// TIA Portal project "Palletizer_TIA_Portal" (V16)

(* hardware
DEVICE "S7-1200 station_1"  S7-1200 Station
   slot 0: "Rack_0"  S7-1200 Rack  Rack  V1.0
   slot 1: "PLC_1"  CPU 1215C DC/DC/DC  6ES7 215-1AG40-0XB0  V4.4
   slot 2: "DI 8x24VDC_1"  6ES7 221-1BF32-0XB0  V2.0
*)

// ===== PLC "PLC_1"  CPU 1215C DC/DC/DC =====

VAR_GLOBAL   // PLC tag table "Tabla de variables estándar"
   "Tag_9" AT %M10.6 : Bool;
   "flanco_p_sensor_entrada_cajas" AT %M10.7 : Bool;
   "Reset_contador_1" AT %M11.0 : Bool;
   "Tag_11" AT %M500.0 : Bool;
   "flanco_p_sensor_ascensor_pales" AT %M11.5 : Bool;
END_VAR

VAR_GLOBAL   // PLC tag table "Entradas"
   "Pallet_at_entry" AT %I0.0 : Bool;   // Sensor al final del transportador de rodillos alimentador, justo antes de la paletizadora
   "Pallet_at_exit" AT %I0.1 : Bool;   // Sensor a la entrada del transportador de rodillos de salida, justo despues de la paletizadora
   "Pallet_loaded" AT %I0.2 : Bool;   // Sensor dentro de la paletizadora, indica que el pale esta dentro
   "Box_at_entry" AT %I0.3 : Bool;   // Sensor al final de la cinta alimentadora de cajas
   "Pusher_limit" AT %I0.4 : Bool;   // Sensor que indica que el empujador esta en alguna de sus posiciones limite
   "Plate_limit" AT %I0.5 : Bool;   // Sensor que indica que la ventana esta en alguna de sus posiciones limite, completamente abierta o completamente cerrada
   "Clamped" AT %I0.6 : Bool;   // Sensor que indica que la mordaza está cerrada
   "Elevator_moving" AT %I0.7 : Bool;   // Sensor que indica que el ascensor está en movimiento
   "Start" AT %I1.0 : Bool;   // Pulsador de start
   "Reset" AT %I1.1 : Bool;   // Pulsador de reset
   "Stop" AT %I1.2 : Bool;   // Pulsador de stop
   "Emergency_stop" AT %I1.3 : Bool;   // Seta de emergencia
   "Auto" AT %I1.4 : Bool;   // Conmutador en modo automatico
   "Manual" AT %I1.5 : Bool;   // Conmutador en modo manual
END_VAR

VAR_GLOBAL   // PLC tag table "Salidas"
   "Pallet_feeder" AT %Q0.0 : Bool;   // Transportador de rodillos alimentador de pales
   "Load_pallet" AT %Q0.1 : Bool;   // Transportador dentro del paletizador
   "Exit_conveyor" AT %Q0.2 : Bool;   // Transportador de rodillos de salida
   "Move_to_limit" AT %Q0.3 : Bool;   // Salida booleana para hacer que la subida o bajada del ascensor sea entre el limite inferior y superior en un solo movimiento
   "Elevator_up" AT %Q0.4 : Bool;   // Ascensor arriba
   "Elevator_down" AT %Q0.5 : Bool;   // Ascensor abajo
   "Box_feeder" AT %Q0.6 : Bool;   // Cinta alimentadora de cajas
   "Turn" AT %Q0.7 : Bool;   // Empujador para girar la caja
   "Push" AT %Q1.0 : Bool;   // Empujador de la caja de la cinta hacia la ventana
   "Load_belt" AT %Q1.1 : Bool;   // Cinta de carga delas cajas dentro del paletizador
   "Clamp" AT %Q1.2 : Bool;   // Mordaza para compactar las cajas
   "Open_plate" AT %Q1.3 : Bool;   // Abrir/cerrar ventana
   "Warning_light" AT %Q1.4 : Bool;   // Luz de peligro
   "Start_light" AT %Q1.5 : Bool;   // Luz de boton de start
   "Reset_light" AT %Q1.6 : Bool;   // Luz de boton de reset
   "Stop_light" AT %Q1.7 : Bool;   // Luz de boton de stop
END_VAR

VAR_GLOBAL   // PLC tag table "variables_en_memoria"
   "Pallet_feeder_manual" AT %M100.0 : Bool;   // Transportador de rodillos alimentador de pales
   "Load_pallet_manual" AT %M100.1 : Bool;   // Transportador dentro del paletizador
   "Exit_conveyor_manual" AT %M100.2 : Bool;   // Transportador de rodillos de salida
   "Move_to_limit_manual" AT %M100.3 : Bool;   // Salida booleana para hacer que la subida o bajada del ascensor sea entre el limite inferior y superior en un solo movimiento
   "Elevator_up_manual" AT %M100.4 : Bool;   // Ascensor arriba
   "Elevator_down_manual" AT %M100.5 : Bool;   // Ascensor abajo
   "Box_feeder_manual" AT %M100.6 : Bool;   // Cinta alimentadora de cajas
   "Turn_manual" AT %M100.7 : Bool;   // Empujador para girar la caja
   "Push_manual" AT %M101.0 : Bool;   // Empujador de la caja de la cinta hacia la ventana
   "Load_belt_manual" AT %M101.1 : Bool;   // Cinta de carga delas cajas dentro del paletizador
   "Clamp_manual" AT %M101.2 : Bool;   // Mordaza para compactar las cajas
   "Open_plate_manual" AT %M101.3 : Bool;   // Abrir/cerrar ventana
   "marcha" AT %M0.0 : Bool;
   "modo_cambiado" AT %M0.1 : Bool;
   "Pallet_terminado" AT %M0.2 : Bool;
   "aux1" AT %M0.3 : Bool;
   "paletizadora_libre" AT %M0.4 : Bool;
   "pale_terminado" AT %M0.5 : Bool;
   "primer_nivel_OK" AT %M0.6 : Bool;
   "segundo_nivel_OK" AT %M0.7 : Bool;
   "flanco_n_sensor_entrada_pales" AT %M10.0 : Bool;
   "flanco_p_sensor_entrada_pales" AT %M10.1 : Bool;
   "flanco_n_sensor_ascensor_pales" AT %M10.3 : Bool;
   "flanco_n_sensor_salida_pales" AT %M10.4 : Bool;
   "flanco_p_sensor_ascensor_pales(1)" AT %M10.5 : Bool;
   "flanco_selector_modo_manual" AT %M200.0 : Bool;
   "flanco_selector_modo_auto" AT %M200.1 : Bool;
   "numero_cajas_1" AT %MW2 : Int;
   "numero_cajas_2" AT %MW4 : Int;
   "numero_columnas-1" AT %MW6 : Int;
   "numero_filas" AT %MW8 : Int;
END_VAR

DATA_BLOCK "control_ascensor_DB"   // DB2
{ S7_Optimized_Access := 'TRUE' }
VERSION : 0.1
// stored: InstanceOfName control_ascensor
"control_ascensor"
BEGIN
END_DATA_BLOCK

DATA_BLOCK "modo_automatico_DB"   // DB3
{ S7_Optimized_Access := 'TRUE' }
VERSION : 0.1
// stored: InstanceOfName modo_automatico
"modo_automatico"
BEGIN
END_DATA_BLOCK

FUNCTION_BLOCK "modo_automatico"   // FB2, LAD
{ S7_Optimized_Access := 'TRUE' }
VERSION : 0.1
   VAR
      E0 : Bool;
      E1 : Bool;
      E2 : Bool;
      E3 : Bool;
      E4 : Bool;
      E5 : Bool;
      "control_roller_1.1" : "control_roller_1";
      "control_roller_2.1" : "control_roller_2";
      control_ascensor_Instance : "control_ascensor";
      control_apilamiento_Instance : "control_apilamiento";
   END_VAR
   VAR_TEMP   // added for the SCL form of the ladder/FBD networks
      _w1 : Bool;
   END_VAR
BEGIN

REGION Network 1
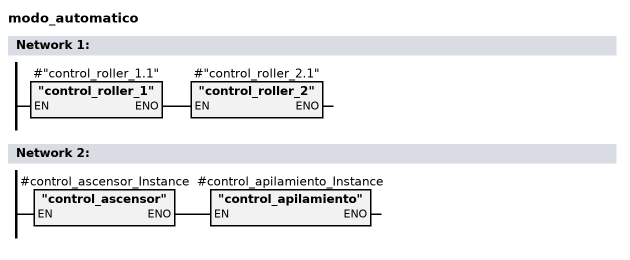
   RUNG wire#powerrail
      #"control_roller_1.1"()
      #"control_roller_2.1"()
   END_RUNG
   // the same network as SCL:
   #"control_roller_1.1"(ENO => #_w1);   // "control_roller_1"
   IF #_w1 THEN
       #"control_roller_2.1"();   // "control_roller_2"
   END_IF;
END_REGION

REGION Network 2
   RUNG wire#powerrail
      #control_ascensor_Instance()
      #control_apilamiento_Instance()
   END_RUNG
   // the same network as SCL:
   #control_ascensor_Instance(ENO => #_w1);   // "control_ascensor"
   IF #_w1 THEN
       #control_apilamiento_Instance();   // "control_apilamiento"
   END_IF;
END_REGION
END_FUNCTION_BLOCK

FUNCTION_BLOCK "control_roller_1"   // FB3, LAD
{ S7_Optimized_Access := 'TRUE' }
VERSION : 0.1
   VAR
      E1 : Bool;
      E2 : Bool;
      E3 : Bool;
      E4 : Bool;
      E5 : Bool;
      E0 : Bool;
   END_VAR
   VAR_TEMP   // added for the SCL form of the ladder/FBD networks
      _w1 : Bool;
      _w2 : Bool;
      _w3 : Bool;
      _w4 : Bool;
   END_VAR
BEGIN

REGION Network 1
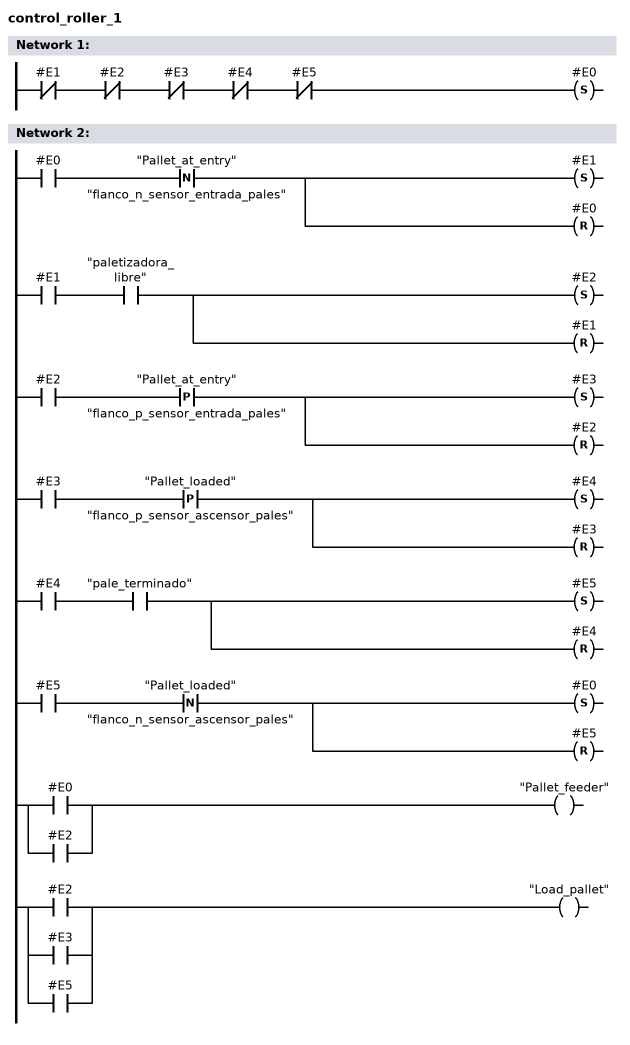
   RUNG wire#powerrail
      I_Contact( #E1 )
      I_Contact( #E2 )
      I_Contact( #E3 )
      I_Contact( #E4 )
      I_Contact( #E5 )
      S_Coil( #E0 )
   END_RUNG
   // the same network as SCL:
   IF NOT #E1 AND NOT #E2 AND NOT #E3 AND NOT #E4 AND NOT #E5 THEN #E0 := TRUE; END_IF;
END_REGION

REGION Network 2
   RUNG wire#powerrail
      Contact( #E0 )
      N_Contact(operand := "Pallet_at_entry", bit := "flanco_n_sensor_entrada_pales")
      wire#w1
      S_Coil( #E1 )
   END_RUNG
   RUNG wire#w1
      R_Coil( #E0 )
   END_RUNG
   RUNG wire#powerrail
      Contact( #E1 )
      Contact( "paletizadora_libre" )
      wire#w2
      S_Coil( #E2 )
   END_RUNG
   RUNG wire#w2
      R_Coil( #E1 )
   END_RUNG
   RUNG wire#powerrail
      Contact( #E2 )
      P_Contact(operand := "Pallet_at_entry", bit := "flanco_p_sensor_entrada_pales")
      wire#w3
      S_Coil( #E3 )
   END_RUNG
   RUNG wire#w3
      R_Coil( #E2 )
   END_RUNG
   RUNG wire#powerrail
      Contact( #E3 )
      P_Contact(operand := "Pallet_loaded", bit := "flanco_p_sensor_ascensor_pales")
      wire#w4
      S_Coil( #E4 )
   END_RUNG
   RUNG wire#w4
      R_Coil( #E3 )
   END_RUNG
   RUNG wire#powerrail
      Contact( #E4 )
      Contact( "pale_terminado" )
      wire#w5
      S_Coil( #E5 )
   END_RUNG
   RUNG wire#w5
      R_Coil( #E4 )
   END_RUNG
   RUNG wire#powerrail
      Contact( #E5 )
      N_Contact(operand := "Pallet_loaded", bit := "flanco_n_sensor_ascensor_pales")
      wire#w6
      S_Coil( #E0 )
   END_RUNG
   RUNG wire#w6
      R_Coil( #E5 )
   END_RUNG
   RUNG wire#powerrail
      Contact( #E0 )
      wire#w7
      Coil( "Pallet_feeder" )
   END_RUNG
   RUNG wire#powerrail
      Contact( #E2 )
   END_RUNG wire#w7
   RUNG wire#powerrail
      Contact( #E2 )
      wire#w8
      Coil( "Load_pallet" )
   END_RUNG
   RUNG wire#powerrail
      Contact( #E3 )
   END_RUNG wire#w8
   RUNG wire#powerrail
      Contact( #E5 )
   END_RUNG wire#w8
   // the same network as SCL:
   #_w1 := #E0 AND NOT "Pallet_at_entry" AND "flanco_n_sensor_entrada_pales";   // falling edge of "Pallet_at_entry"
   "flanco_n_sensor_entrada_pales" := "Pallet_at_entry";
   IF #_w1 THEN
       #E1 := TRUE;
       #E0 := FALSE;
   END_IF;
   IF #E1 AND "paletizadora_libre" THEN
       #E2 := TRUE;
       #E1 := FALSE;
   END_IF;
   #_w2 := #E2 AND "Pallet_at_entry" AND NOT "flanco_p_sensor_entrada_pales";   // rising edge of "Pallet_at_entry"
   "flanco_p_sensor_entrada_pales" := "Pallet_at_entry";
   IF #_w2 THEN
       #E3 := TRUE;
       #E2 := FALSE;
   END_IF;
   #_w3 := #E3 AND "Pallet_loaded" AND NOT "flanco_p_sensor_ascensor_pales";   // rising edge of "Pallet_loaded"
   "flanco_p_sensor_ascensor_pales" := "Pallet_loaded";
   IF #_w3 THEN
       #E4 := TRUE;
       #E3 := FALSE;
   END_IF;
   IF #E4 AND "pale_terminado" THEN
       #E5 := TRUE;
       #E4 := FALSE;
   END_IF;
   #_w4 := #E5 AND NOT "Pallet_loaded" AND "flanco_n_sensor_ascensor_pales";   // falling edge of "Pallet_loaded"
   "flanco_n_sensor_ascensor_pales" := "Pallet_loaded";
   IF #_w4 THEN
       #E0 := TRUE;
       #E5 := FALSE;
   END_IF;
   "Pallet_feeder" := #E0 OR #E2;
   "Load_pallet" := #E2 OR #E3 OR #E5;
END_REGION
END_FUNCTION_BLOCK

FUNCTION_BLOCK "control_roller_2"   // FB4, LAD
{ S7_Optimized_Access := 'TRUE' }
VERSION : 0.1
   VAR
      Timer_TP_1 : TP_TIME;
   END_VAR
   VAR_TEMP   // added for the SCL form of the ladder/FBD networks
      _w1 : Bool;
   END_VAR
BEGIN

REGION Network 1: Transportador de rodillos de salida
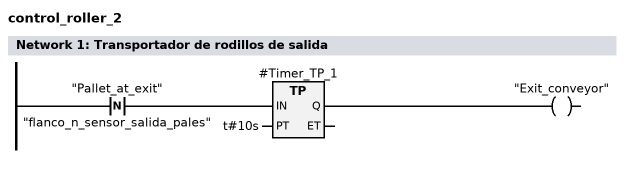
   #_w1 := NOT "Pallet_at_exit" AND "flanco_n_sensor_salida_pales";   // falling edge of "Pallet_at_exit"
   "flanco_n_sensor_salida_pales" := "Pallet_at_exit";
   #Timer_TP_1(IN := #_w1, PT := t#10s);   // TP
   "Exit_conveyor" := #Timer_TP_1.Q;
END_REGION
END_FUNCTION_BLOCK

FUNCTION_BLOCK "control_ascensor"   // FB5, LAD
{ S7_Optimized_Access := 'TRUE' }
VERSION : 0.1
   VAR
      E0 : Bool;
      E1 : Bool;
      E2 : Bool;
      E3 : Bool;
      E4 : Bool;
      E5 : Bool;
      E6 : Bool;
      TON_instancia_1 : TON_TIME;
      TON_instancia_2 : TON_TIME;
      TON_instancia_3 : TON_TIME;
   END_VAR
   VAR_TEMP   // added for the SCL form of the ladder/FBD networks
      _w1 : Bool;
      _w2 : Bool;
      _w3 : Bool;
      _w4 : Bool;
   END_VAR
BEGIN

REGION Network 1
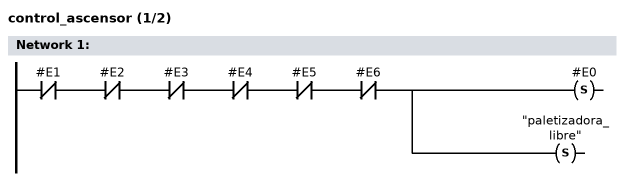
   RUNG wire#powerrail
      I_Contact( #E1 )
      I_Contact( #E2 )
      I_Contact( #E3 )
      I_Contact( #E4 )
      I_Contact( #E5 )
      I_Contact( #E6 )
      wire#w1
      S_Coil( #E0 )
   END_RUNG
   RUNG wire#w1
      S_Coil( "paletizadora_libre" )
   END_RUNG
   // the same network as SCL:
   IF NOT #E1 AND NOT #E2 AND NOT #E3 AND NOT #E4 AND NOT #E5 AND NOT #E6 THEN
       #E0 := TRUE;
       "paletizadora_libre" := TRUE;
   END_IF;
END_REGION

REGION Network 2: Salida booleana para hacer que la subida o bajada del ascensor sea entre el limite inferior y superior en un solo movimiento
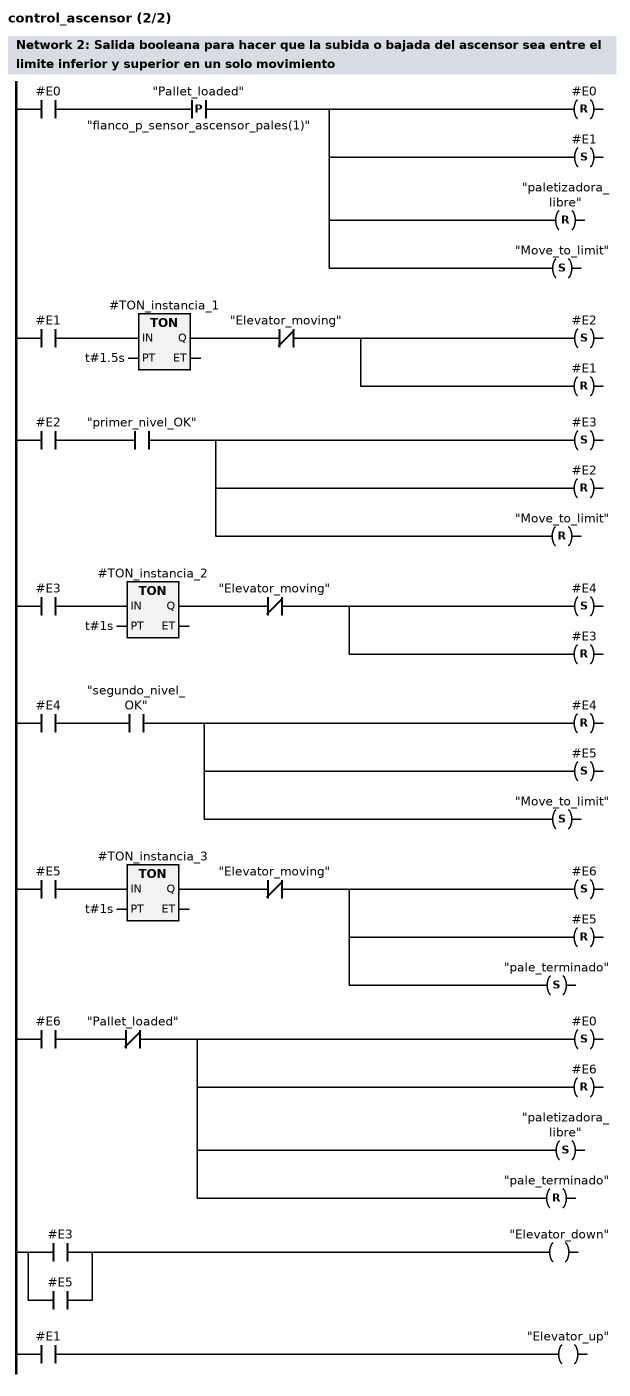
   #_w1 := #E0 AND "Pallet_loaded" AND NOT "flanco_p_sensor_ascensor_pales(1)";   // rising edge of "Pallet_loaded"
   "flanco_p_sensor_ascensor_pales(1)" := "Pallet_loaded";
   IF #_w1 THEN
       #E0 := FALSE;
       #E1 := TRUE;
       "paletizadora_libre" := FALSE;
       "Move_to_limit" := TRUE;
   END_IF;
   #TON_instancia_1(IN := #E1, PT := t#1.5s);   // TON
   IF #TON_instancia_1.Q AND NOT "Elevator_moving" THEN
       #E2 := TRUE;
       #E1 := FALSE;
   END_IF;
   IF #E2 AND "primer_nivel_OK" THEN #E3 := TRUE; END_IF;
   #_w2 := #E2 AND "primer_nivel_OK";
   IF #_w2 THEN
       #E2 := FALSE;
       "Move_to_limit" := FALSE;
   END_IF;
   #TON_instancia_2(IN := #E3, PT := t#1s);   // TON
   IF #TON_instancia_2.Q AND NOT "Elevator_moving" THEN
       #E4 := TRUE;
       #E3 := FALSE;
   END_IF;
   #_w3 := #E4 AND "segundo_nivel_OK";
   IF #_w3 THEN
       #E4 := FALSE;
       #E5 := TRUE;
       "Move_to_limit" := TRUE;
   END_IF;
   #TON_instancia_3(IN := #E5, PT := t#1s);   // TON
   IF #TON_instancia_3.Q AND NOT "Elevator_moving" THEN
       #E6 := TRUE;
       #E5 := FALSE;
       "pale_terminado" := TRUE;
   END_IF;
   IF #E6 AND NOT "Pallet_loaded" THEN #E0 := TRUE; END_IF;
   #_w4 := #E6 AND NOT "Pallet_loaded";
   IF #_w4 THEN
       #E6 := FALSE;
       "paletizadora_libre" := TRUE;
       "pale_terminado" := FALSE;
   END_IF;
   "Elevator_down" := #E3 OR #E5;
   "Elevator_up" := #E1;
END_REGION
END_FUNCTION_BLOCK

FUNCTION_BLOCK "control_apilamiento"   // FB6, LAD
{ S7_Optimized_Access := 'TRUE' }
VERSION : 0.1
   VAR
      E0 : Bool;
      E1 : Bool;
      E2 : Bool;
      E3 : Bool;
      E4 : Bool;
      E5 : Bool;
      E6 : Bool;
      E7 : Bool;
      E8 : Bool;
      E9 : Bool;
   END_VAR
   VAR RETAIN
      CTU_1 : CTD_INT;
   END_VAR
   VAR
      TON_1 : TON_TIME;
      TON_2 : TON_TIME;
      TON_3 : TON_TIME;
   END_VAR
   VAR RETAIN
      CTU_2 : CTU_INT;
   END_VAR
   VAR
      TON_4 : TON_TIME;
      TON_5 : TON_TIME;
      TON_6 : TON_TIME;
      TON_7 : TON_TIME;
      TON_8 : TON_TIME;
   END_VAR
   VAR_TEMP   // added for the SCL form of the ladder/FBD networks
      _w1 : Bool;
      _w2 : Bool;
      _w3 : Bool;
      _w4 : Bool;
   END_VAR
BEGIN

REGION Network 1
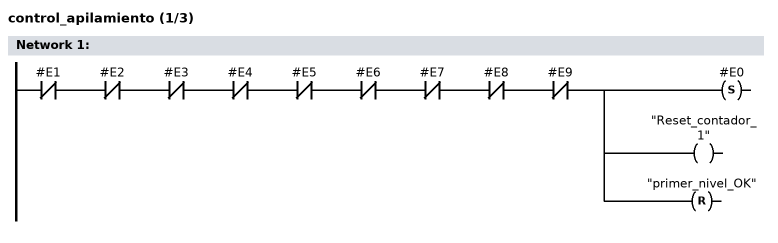
   RUNG wire#powerrail
      I_Contact( #E1 )
      I_Contact( #E2 )
      I_Contact( #E3 )
      I_Contact( #E4 )
      I_Contact( #E5 )
      I_Contact( #E6 )
      I_Contact( #E7 )
      I_Contact( #E8 )
      I_Contact( #E9 )
      wire#w1
      S_Coil( #E0 )
   END_RUNG
   RUNG wire#w1
      Coil( "Reset_contador_1" )
   END_RUNG
   RUNG wire#w1
      R_Coil( "primer_nivel_OK" )
   END_RUNG
   // the same network as SCL:
   #_w1 := NOT #E1 AND NOT #E2 AND NOT #E3 AND NOT #E4 AND NOT #E5 AND NOT #E6 AND NOT #E7 AND NOT #E8 AND NOT #E9;
   IF #_w1 THEN #E0 := TRUE; END_IF;
   "Reset_contador_1" := #_w1;
   IF #_w1 THEN "primer_nivel_OK" := FALSE; END_IF;
END_REGION

REGION Network 2
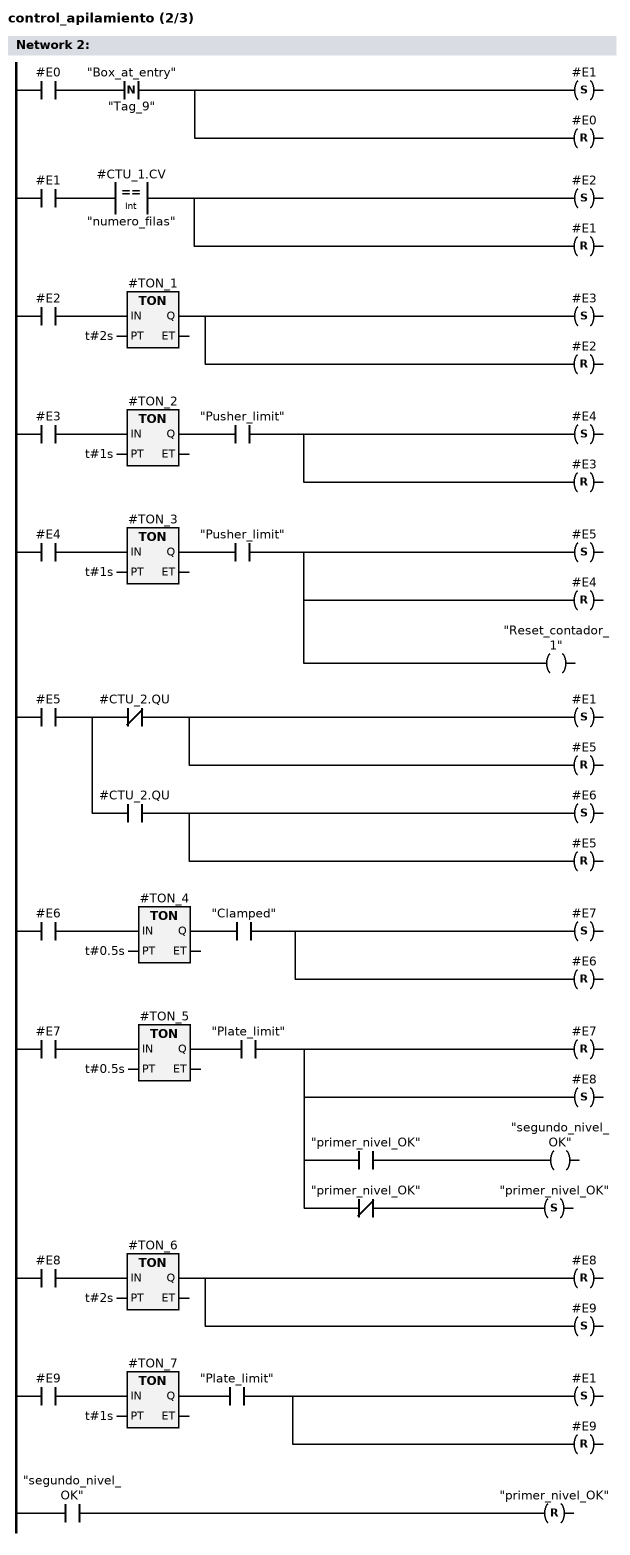
   #_w1 := #E0 AND NOT "Box_at_entry" AND "Tag_9";   // falling edge of "Box_at_entry"
   "Tag_9" := "Box_at_entry";
   IF #_w1 THEN
       #E1 := TRUE;
       #E0 := FALSE;
   END_IF;
   IF #E1 AND (#CTU_1.CV = "numero_filas") THEN
       #E2 := TRUE;
       #E1 := FALSE;
   END_IF;
   #TON_1(IN := #E2, PT := t#2s);   // TON
   IF #TON_1.Q THEN
       #E3 := TRUE;
       #E2 := FALSE;
   END_IF;
   #TON_2(IN := #E3, PT := t#1s);   // TON
   IF #TON_2.Q AND "Pusher_limit" THEN
       #E4 := TRUE;
       #E3 := FALSE;
   END_IF;
   #TON_3(IN := #E4, PT := t#1s);   // TON
   #_w2 := #TON_3.Q AND "Pusher_limit";
   IF #_w2 THEN
       #E5 := TRUE;
       #E4 := FALSE;
   END_IF;
   "Reset_contador_1" := #_w2;
   IF #E5 AND NOT #CTU_2.QU THEN #E1 := TRUE; END_IF;
   #_w3 := #E5;
   IF #E5 AND NOT #CTU_2.QU THEN #E5 := FALSE; END_IF;
   IF #_w3 AND #CTU_2.QU THEN
       #E6 := TRUE;
       #E5 := FALSE;
   END_IF;
   #TON_4(IN := #E6, PT := t#0.5s);   // TON
   IF #TON_4.Q AND "Clamped" THEN
       #E7 := TRUE;
       #E6 := FALSE;
   END_IF;
   #TON_5(IN := #E7, PT := t#0.5s);   // TON
   #_w4 := #TON_5.Q AND "Plate_limit";
   IF #_w4 THEN
       #E7 := FALSE;
       #E8 := TRUE;
   END_IF;
   "segundo_nivel_OK" := #_w4 AND "primer_nivel_OK";
   IF #_w4 AND NOT "primer_nivel_OK" THEN "primer_nivel_OK" := TRUE; END_IF;
   #TON_6(IN := #E8, PT := t#2s);   // TON
   IF #TON_6.Q THEN
       #E8 := FALSE;
       #E9 := TRUE;
   END_IF;
   #TON_7(IN := #E9, PT := t#1s);   // TON
   IF #TON_7.Q AND "Plate_limit" THEN
       #E1 := TRUE;
       #E9 := FALSE;
   END_IF;
   IF "segundo_nivel_OK" THEN "primer_nivel_OK" := FALSE; END_IF;
END_REGION

REGION Network 3: Cinta alimentadora de cajas
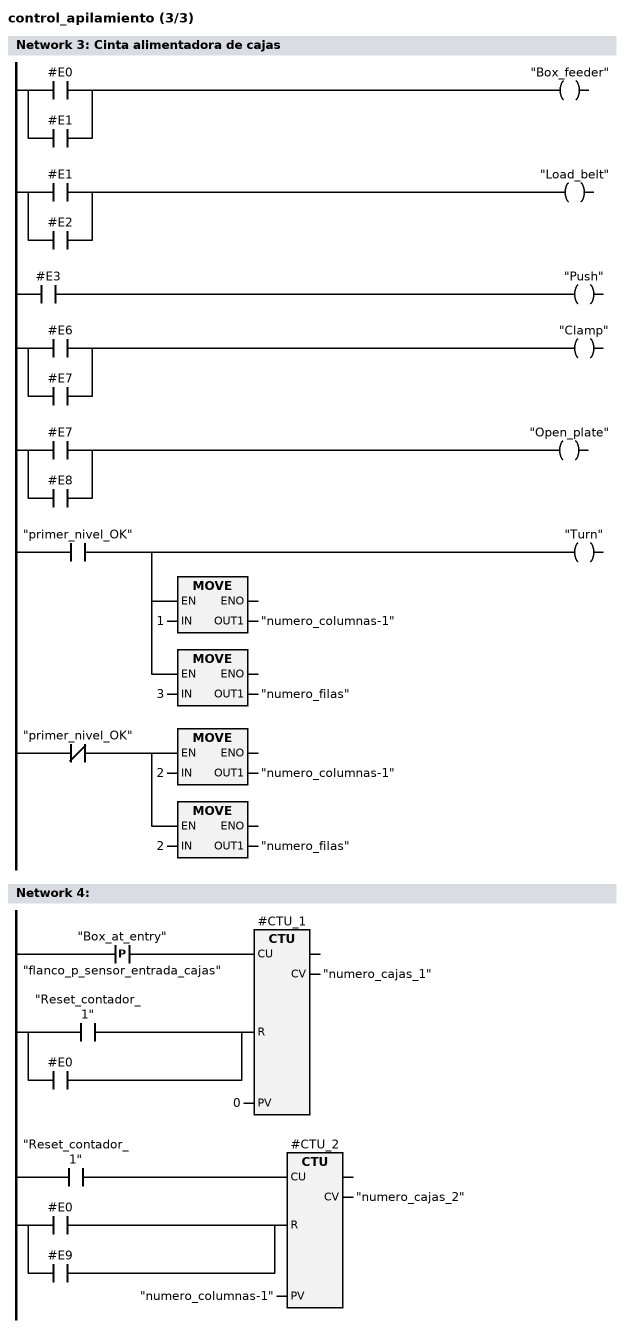
   RUNG wire#powerrail
      Contact( #E0 )
      wire#w1
      Coil( "Box_feeder" )
   END_RUNG
   RUNG wire#powerrail
      Contact( #E1 )
   END_RUNG wire#w1
   RUNG wire#powerrail
      Contact( #E1 )
      wire#w2
      Coil( "Load_belt" )
   END_RUNG
   RUNG wire#powerrail
      Contact( #E2 )
   END_RUNG wire#w2
   RUNG wire#powerrail
      Contact( #E3 )
      Coil( "Push" )
   END_RUNG
   RUNG wire#powerrail
      Contact( #E6 )
      wire#w3
      Coil( "Clamp" )
   END_RUNG
   RUNG wire#powerrail
      Contact( #E7 )
   END_RUNG wire#w3
   RUNG wire#powerrail
      Contact( #E7 )
      wire#w4
      Coil( "Open_plate" )
   END_RUNG
   RUNG wire#powerrail
      Contact( #E8 )
   END_RUNG wire#w4
   RUNG wire#powerrail
      Contact( "primer_nivel_OK" )
      wire#w5
      Coil( "Turn" )
   END_RUNG
   RUNG wire#w5
      Move(in := 1, out1 => "numero_columnas-1")
   END_RUNG
   RUNG wire#w5
      Move(in := 3, out1 => "numero_filas")
   END_RUNG
   RUNG wire#powerrail
      I_Contact( "primer_nivel_OK" )
      wire#w6
      Move(in := 2, out1 => "numero_columnas-1")
   END_RUNG
   RUNG wire#w6
      Move(in := 2, out1 => "numero_filas")
   END_RUNG
   // the same network as SCL:
   "Box_feeder" := #E0 OR #E1;
   "Load_belt" := #E1 OR #E2;
   "Push" := #E3;
   "Clamp" := #E6 OR #E7;
   "Open_plate" := #E7 OR #E8;
   "Turn" := "primer_nivel_OK";
   IF "primer_nivel_OK" THEN
       "numero_columnas-1" := 1;
       "numero_filas" := 3;
   END_IF;
   IF NOT "primer_nivel_OK" THEN
       "numero_columnas-1" := 2;
       "numero_filas" := 2;
   END_IF;
END_REGION

REGION Network 4
   #_w1 := "Box_at_entry" AND NOT "flanco_p_sensor_entrada_cajas";   // rising edge of "Box_at_entry"
   "flanco_p_sensor_entrada_cajas" := "Box_at_entry";
   #CTU_1(CU := #_w1, R := "Reset_contador_1" OR #E0, PV := 0, CV => "numero_cajas_1");   // CTU
   #CTU_2(CU := "Reset_contador_1", R := #E0 OR #E9, PV := "numero_columnas-1", CV => "numero_cajas_2");   // CTU
END_REGION
END_FUNCTION_BLOCK

ORGANIZATION_BLOCK "Main"   // OB1, LAD, ProgramCycle
TITLE = "Main Program Sweep (Cycle)"
{ S7_Optimized_Access := 'TRUE' }
VERSION : 0.1
   VAR_INPUT
      Initial_Call : Bool;   // Initial call of this OB
      Remanence : Bool;   // =True, if remanent data are available
   END_VAR
   VAR_TEMP   // added for the SCL form of the ladder/FBD networks
      _w1 : Bool;
      _w2 : Bool;
   END_VAR
BEGIN

REGION Network 1
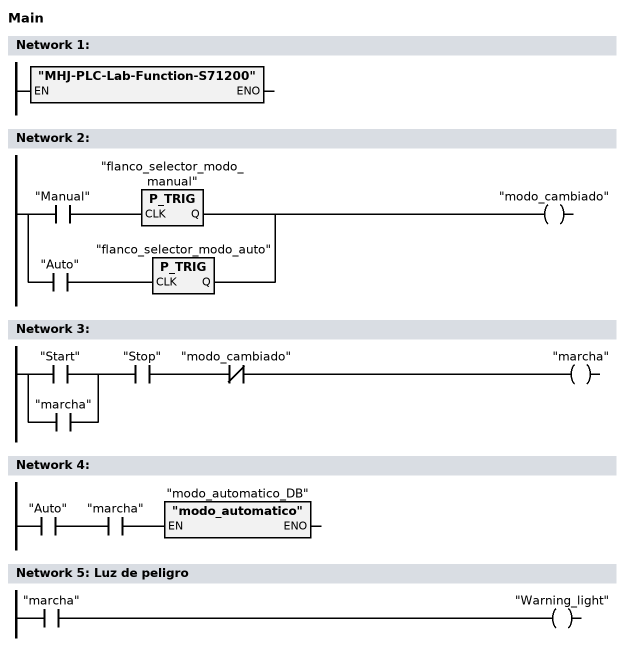
   RUNG wire#powerrail
      "MHJ-PLC-Lab-Function-S71200"()
   END_RUNG
   // the same network as SCL:
   "MHJ-PLC-Lab-Function-S71200"();
END_REGION

REGION Network 2
   RUNG wire#powerrail
      Contact( "Manual" )
      P_Trig( "flanco_selector_modo_manual" )
      wire#w1
      Coil( "modo_cambiado" )
   END_RUNG
   RUNG wire#powerrail
      Contact( "Auto" )
      P_Trig( "flanco_selector_modo_auto" )
   END_RUNG wire#w1
   // the same network as SCL:
   #_w1 := "Manual" AND NOT "flanco_selector_modo_manual";   // rising edge
   "flanco_selector_modo_manual" := "Manual";
   #_w2 := "Auto" AND NOT "flanco_selector_modo_auto";   // rising edge
   "flanco_selector_modo_auto" := "Auto";
   "modo_cambiado" := #_w1 OR #_w2;
END_REGION

REGION Network 3
   RUNG wire#powerrail
      Contact( "Start" )
      wire#w1
      Contact( "Stop" )
      I_Contact( "modo_cambiado" )
      Coil( "marcha" )
   END_RUNG
   RUNG wire#powerrail
      Contact( "marcha" )
   END_RUNG wire#w1
   // the same network as SCL:
   "marcha" := ("Start" OR "marcha") AND "Stop" AND NOT "modo_cambiado";
END_REGION

REGION Network 4
   RUNG wire#powerrail
      Contact( "Auto" )
      Contact( "marcha" )
      "modo_automatico_DB"()
   END_RUNG
   // the same network as SCL:
   IF "Auto" AND "marcha" THEN
       "modo_automatico_DB"();   // "modo_automatico"
   END_IF;
END_REGION

REGION Network 5: Luz de peligro
   RUNG wire#powerrail
      Contact( "marcha" )
      Coil( "Warning_light" )
   END_RUNG
   // the same network as SCL:
   "Warning_light" := "marcha";
END_REGION
END_ORGANIZATION_BLOCK

// folder: conexion_factoryIO

FUNCTION "MHJ-PLC-Lab-Function-S71200" : Void   // FC9000, SCL
{ S7_Optimized_Access := 'TRUE' }
VERSION : 0.1
   VAR_TEMP
      rdTimeReturn : Int;
      outputTime : DTL;
      SyncVal : Byte;
      forVal : Int;
      forVal_2 : Int;
      Value : Byte;
   END_VAR
   VAR CONSTANT
      CompVal : Byte := 16#34;
      Value_01 : Byte := 16#11;
      Value_01_DW : DWord := 16#A165_D992;
      Value_02_DW : DWord := 16#58BE_4401;
   END_VAR
BEGIN

   #Value:=PEEK(area := 16#82,
        dbNumber := 0,
        byteOffset := 511);
   #Value := #Value + 1;

   POKE(area := 16#82,
        dbNumber := 0,
        byteOffset := 511,
        value := #Value);

   POKE(area:=16#81,
        dbNumber:=0,
        byteOffset:=1016,
        value:=#Value_01_DW);
   POKE(area := 16#81,
        dbNumber := 0,
        byteOffset := 1020,
        value := #Value_02_DW);

   POKE(area := 16#81,
        dbNumber := 0,
        byteOffset := 511,
        value := B#16#00);

   FOR #forVal := 0 TO 120 DO
       FOR #forVal_2:=0 TO 10 DO
           #rdTimeReturn:=RD_SYS_T(#outputTime);
           #rdTimeReturn := WR_SYS_T(#outputTime);
           #rdTimeReturn := RD_SYS_T(#outputTime);
           #rdTimeReturn := WR_SYS_T(#outputTime);
       END_FOR;
       #SyncVal:= PEEK(area := 16#81,
                      dbNumber := 0,
                      byteOffset := 511);
       IF #SyncVal = #CompVal THEN
          GOTO M_1;
       END_IF;
   END_FOR;
   RETURN;

   M_1:
   POKE(area := 16#81,
        dbNumber := 0,
        byteOffset := 511,
        value := B#16#0);
END_FUNCTION